INTERFACE I_ChunkedRequestData EXTENDS I_SessionData

PROPERTY PUBLIC IsComplete : BOOL
GET
END_GET
END_PROPERTY

PROPERTY PUBLIC PayloadAddress : POINTER TO STRING
GET
END_GET
END_PROPERTY

PROPERTY PUBLIC PayloadSizeInBytes : UDINT
GET
END_GET
END_PROPERTY

METHOD PUBLIC TryAddChunkedPayload : BOOL;
VAR_INPUT
	PayloadAddress : POINTER TO STRING;
	PayloadSize : UDINT;
	ChunkSequence : DINT;
END_VAR
END_METHOD

END_INTERFACE

(* stored: Version 1.1.0.1, ProductVersion 3.1.4024.13
   Itf I_ChunkedRequestData: Id {d6d9650a-3b8f-0f35-30e2-315a5480f9d9}
   Property IsComplete: Id {05254a89-32fd-0863-364a-f86b5302016e}
   Get Get: Id {c73ea561-9454-0512-1793-f1afca724b37}
   Property PayloadAddress: Id {3f79f664-186a-00c1-3063-4fe27b637d8f}
   Get Get: Id {d44e22f6-668d-0d57-1862-de4d030f68c0}
   Property PayloadSizeInBytes: Id {5854569a-304a-0faa-35b5-a0b581a26e4c}
   Get Get: Id {766b1610-02ec-0fe6-087b-42d53cd45cae}
   Method TryAddChunkedPayload: Id {a2456111-d73b-02d0-0426-e73fdc45cea9} *)
